// TIA Portal project "机制231陈煜暄2026621" (V15)

(* hardware
DEVICE "HMI_1"  KTP700 Basic PN
   slot 0: "HMI_1"  KTP700 Basic PN  6AV2 123-2GB03-0AX0  15.0.0.0
   slot 1: "HMI_RT_1"  KTP700 Basic PN  6AV2 123-2GB03-0AX0  15.0.0.0
   slot 5: "HMI_1.IE_CP_1"  PROFINET Interface  15.0.0.0
      slot 1: "PROFINET Interface_1"  PROFINET Interface
         slot 1: "Port_1"  Port
DEVICE "S7-1200 station_1"  S7-1200 Station
   slot 0: "Rack_0"  S7-1200 Rack  Rack  V1.0
   slot 1: "PLC_1"  CPU 1214C DC/DC/DC  6ES7 214-1AG40-0XB0  V4.2
*)

// ===== PLC "PLC_1"  CPU 1214C DC/DC/DC =====

VAR_GLOBAL   // PLC tag table "默认变量表"
   "复位" AT %I0.2 : Bool;
   "切换快" AT %I0.7 : Bool;
   "切换慢" AT %I1.0 : Bool;
   "开始" AT %I1.1 : Bool;
   "停止" AT %I1.2 : Bool;
   "气缸1伸出" AT %Q0.6 : Bool;
   "气缸2伸出" AT %Q0.7 : Bool;
   "气缸2缩回" AT %Q1.0 : Bool;
   "气缸1缩回" AT %Q1.1 : Bool;
END_VAR

DATA_BLOCK "气缸"   // DB1
{ S7_Optimized_Access := 'TRUE' }
VERSION : 0.1
   VAR
      启动 : Bool;
      停止 : Bool;
      复位 : Bool;
      气缸运行 : Bool;
      步骤 : Int;
      频率 : Time := T#1s;
      计时器1 : TON_TIME;
      计时器2 : TON_TIME;
      计时器3 : TON_TIME;
      计时器4 : TON_TIME;
      流水灯1 : Bool;
      流水灯2 : Bool;
      流水灯3 : Bool;
   END_VAR
BEGIN
END_DATA_BLOCK

ORGANIZATION_BLOCK "Main"   // OB1, LAD, ProgramCycle
TITLE = "Main Program Sweep (Cycle)"
{ S7_Optimized_Access := 'TRUE' }
VERSION : 0.1
   VAR_INPUT
      Initial_Call : Bool;   // Initial call of this OB
      Remanence : Bool;   // =True, if remanent data are available
   END_VAR
   VAR_TEMP   // added for the SCL form of the ladder/FBD networks
      _w1 : Bool;
   END_VAR
BEGIN

REGION Network 1: 控制流动
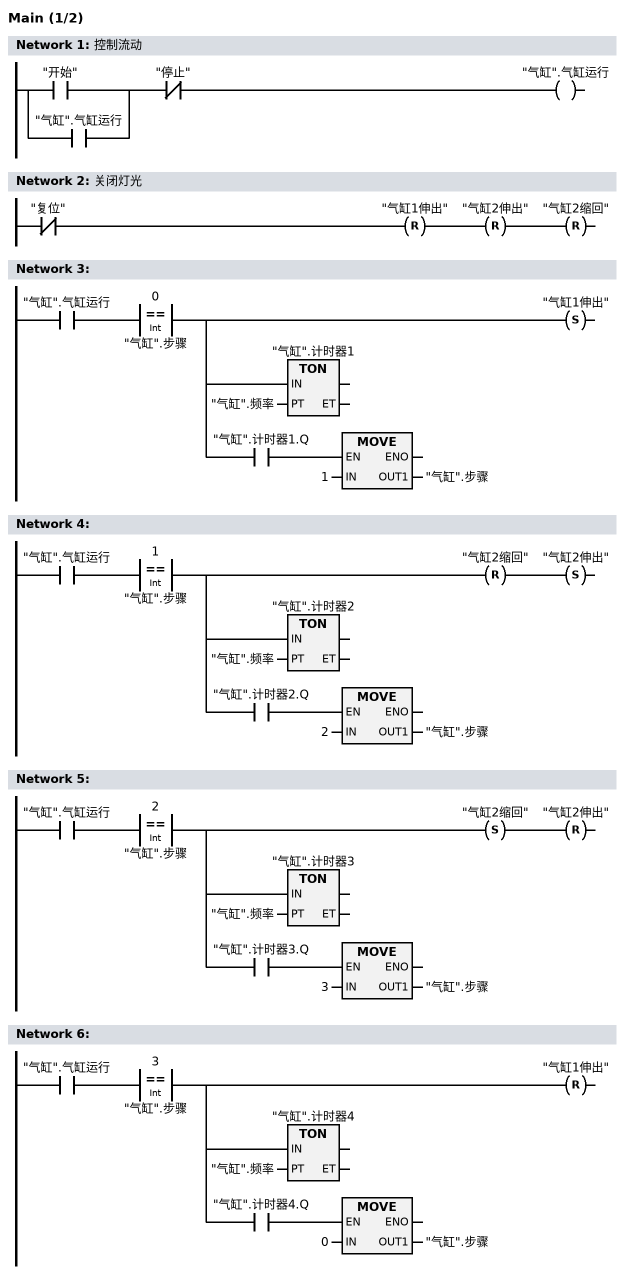
   RUNG wire#powerrail
      Contact( "开始" )
      wire#w1
      I_Contact( "停止" )
      Coil( "气缸".气缸运行 )
   END_RUNG
   RUNG wire#powerrail
      Contact( "气缸".气缸运行 )
   END_RUNG wire#w1
   // the same network as SCL:
   "气缸".气缸运行 := ("开始" OR "气缸".气缸运行) AND NOT "停止";
END_REGION

REGION Network 2: 关闭灯光
   RUNG wire#powerrail
      I_Contact( "复位" )
      R_Coil( "气缸1伸出" )
      R_Coil( "气缸2伸出" )
      R_Coil( "气缸2缩回" )
   END_RUNG
   // the same network as SCL:
   IF NOT "复位" THEN
       "气缸1伸出" := FALSE;
       "气缸2伸出" := FALSE;
       "气缸2缩回" := FALSE;
   END_IF;
END_REGION

REGION Network 3
   #_w1 := "气缸".气缸运行 AND (0 = "气缸".步骤);
   IF #_w1 THEN "气缸1伸出" := TRUE; END_IF;
   "气缸".计时器1.TON(IN := #_w1, PT := "气缸".频率);
   IF #_w1 AND "气缸".计时器1.Q THEN "气缸".步骤 := 1; END_IF;
END_REGION

REGION Network 4
   #_w1 := "气缸".气缸运行 AND (1 = "气缸".步骤);
   IF #_w1 THEN
       "气缸2缩回" := FALSE;
       "气缸2伸出" := TRUE;
   END_IF;
   "气缸".计时器2.TON(IN := #_w1, PT := "气缸".频率);
   IF #_w1 AND "气缸".计时器2.Q THEN "气缸".步骤 := 2; END_IF;
END_REGION

REGION Network 5
   #_w1 := "气缸".气缸运行 AND (2 = "气缸".步骤);
   IF #_w1 THEN
       "气缸2缩回" := TRUE;
       "气缸2伸出" := FALSE;
   END_IF;
   "气缸".计时器3.TON(IN := #_w1, PT := "气缸".频率);
   IF #_w1 AND "气缸".计时器3.Q THEN "气缸".步骤 := 3; END_IF;
END_REGION

REGION Network 6
   #_w1 := "气缸".气缸运行 AND (3 = "气缸".步骤);
   IF #_w1 THEN "气缸1伸出" := FALSE; END_IF;
   "气缸".计时器4.TON(IN := #_w1, PT := "气缸".频率);
   IF #_w1 AND "气缸".计时器4.Q THEN "气缸".步骤 := 0; END_IF;
END_REGION

REGION Network 7: 0
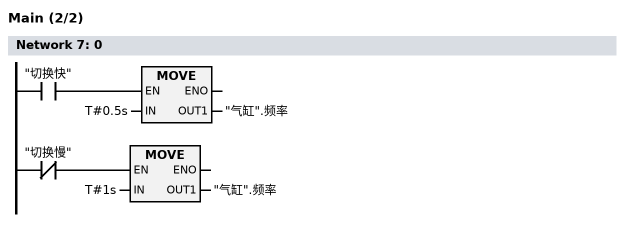
   RUNG wire#powerrail
      Contact( "切换快" )
      Move(in := T#0.5s, out1 => "气缸".频率)
   END_RUNG
   RUNG wire#powerrail
      I_Contact( "切换慢" )
      Move(in := T#1s, out1 => "气缸".频率)
   END_RUNG
   // the same network as SCL:
   IF "切换快" THEN "气缸".频率 := T#0.5s; END_IF;
   IF NOT "切换慢" THEN "气缸".频率 := T#1s; END_IF;
END_REGION
END_ORGANIZATION_BLOCK

(* ===== HMI "HMI_RT_1" =====
system functions are stored by id; their names below are inferred from use
connection "HMI_连接_1": ETHERNET, SMART_S7_1200_OMS

HMI tags "默认变量表"
   "Tag_ScreenNumber" : UInt, internal
   "流水灯_启动" : Bool = PLC 气缸.启动, 1 s
   "流水灯_停止" : Bool = PLC 气缸.停止, 1 s
   "流水灯_复位" : Bool = PLC 气缸.复位, 1 s
   "流水灯_流水灯1" : Bool = PLC 气缸.流水灯1, 1 s
   "流水灯_流水灯2" : Bool = PLC 气缸.流水灯2, 1 s
   "流水灯_流水灯3" : Bool = PLC 气缸.流水灯3, 1 s

Template "Template_1" 800x480
   Button "退出" at 714,429 size 71x50; TextOff '退出'; PictureOff "ExitRuntime_KTP700_Basic_PN_TR"; PictureOn "ExitRuntime_KTP700_Basic_PN_TR"
      on Release: StopRuntime(0)
   Button "Template_Button" at 614,429 size 71x50; TextOff 'Text'
   Button "Template_Button_1" at 514,429 size 71x50; TextOff 'Text'
   Button "Template_Button_2" at 414,429 size 71x50; TextOff 'Text'
   Button "Template_Button_3" at 314,429 size 71x50; TextOff 'Text'
   Button "Template_Button_4" at 214,429 size 71x50; TextOff 'Text'
   Button "报警" at 114,429 size 71x50; TextOff '报警'; PictureOff "AlarmDisplay_KTP700_Basic_PN_TR"; PictureOn "AlarmDisplay_KTP700_Basic_PN_TR"
      on Release: function_ef3f5d25("报警窗口_Unacknowledged", -1)
   Button "起始画面" at 14,429 size 71x50; TextOff '起始画面'; PictureOff "NavigateHome_KTP700_Basic_PN_TR"; PictureOn "NavigateHome_KTP700_Basic_PN_TR"
      on Release: ActivateScreen("根画面", 0)
   SymbolicIOField "Symbolic_IO_Field_Screen" at 93,9 size 600x33; TextOff '0'; TextOn '1'; TextList "TextList_ScreenNames"
      ProcessValue <- "Tag_ScreenNumber"
      on Change: ActivateScreenByNumber("Tag_ScreenNumber", 0)
   DateTimeField "HmiScreenItemData" at 695,25 size 105x25
   DateTimeField "HmiScreenItemData_1" at 695,0 size 105x25
   GraphicView "Logo" at 0,0 size 91x51; Picture "HMI_1 的 Logo"

screen "根画面" 800x480, template "Template_1"
   on GenerateScreen: SetTag("Tag_ScreenNumber", 1)
   TextField "HmiScreenItemData" at 75,42 size 640x25; Text '欢迎进入 HMI_1 (KTP700 Basic+ PN)！'
   Circle "圆_1" at 415,168 size 48x48
      Appearance <- "流水灯_流水灯1"
   Button "按钮_1" at 108,121 size 95x47; TextOff '启动'
      on Press: SetBit("流水灯_启动")
      on Release: ResetBit("流水灯_启动")
   Button "按钮_2" at 229,123 size 95x47; TextOff '停止'
      on Release: ResetBit("流水灯_停止")
      on Press: SetBit("流水灯_停止")
   Button "按钮_3" at 108,190 size 95x47; TextOff '复位'
      on Release: ResetBit("流水灯_复位")
      on Press: SetBit("流水灯_复位")
   Circle "圆_2" at 491,170 size 48x48
      Appearance <- "流水灯_流水灯2"
   Circle "圆_3" at 573,170 size 48x48
      Appearance <- "流水灯_流水灯3"
*)